// TIA Portal V19 export
DATA_BLOCK "UP_CM03.GP03"   // DB1003
// stored: AutoNumber false, InstanceOfName UP_Spuele.GP0x, InstanceOfType FB
"UP_Spuele.GP0x"
   // VAR RETAIN
   //    In { ExternalAccessible := 'False'; ExternalVisible := 'False'; ExternalWritable := 'False'} : Struct
   //       NotHalt : Bool;
   //       ext_Freigabe : Bool;
   //       TW_senkt : Bool;
   //       Auto : Bool;
   //       Ein : Bool;
   //       FU_betriebsbereit : Bool;
   //       FU_Stoerung : Bool;
   //       Niv_TLS : Bool;
   //       Niv_min : Bool;
   //       Frg_Niv_CM05 : Bool;
   //       SRM_Saugseite_auf : Bool;
   //       SRM_Saugseite_zu : Bool;
   //       SRM_Druckseite_auf : Bool;
   //       SRM_Druckseite_zu : Bool;
   //       GW_p_UP : Bool;
   //       Betriebsart : USInt;
   //       FU_speed : Int;
   //       Druck_Pumpe : Real;
   //    END_STRUCT;
   //    Param { ExternalAccessible := 'False'; ExternalVisible := 'False'; ExternalWritable := 'False'} : Struct
   //       SW_Hand : Int;
   //       SW_Auto_AZ : Int;
   //       SW_Auto_aAZ : Int;
   //       Spülzeit : Time;
   //       DT_Druckaufbau : Time;
   //       DT_Testzeit : Time;
   //       SW_Drucktest : Real;
   //       "Name" : String[12];
   //    END_STRUCT;
   //    Zst { ExternalAccessible := 'False'; ExternalVisible := 'False'; ExternalWritable := 'False'} : Struct
   //       Niveau : USInt;
   //       Status_GP0x : USInt;
   //       Status_DT : USInt;
   //       Restzeit_Spülen : Time;
   //       Restzeit_DT : Time;
   //       TON_Spülventil_auf : Bool;
   //       Spuelen : Bool;
   //       Spuelen_aktiv : Bool;
   //       Drucktest_aktiv : Bool;
   //       Umwaelzen : Bool;
   //       Zeit_laeuft : Bool;
   //       Drucktest_ok : Bool;
   //       Bedienung_erlaubt : Bool;
   //       speed : Int;
   //    END_STRUCT;
   //    Mld { ExternalAccessible := 'False'; ExternalVisible := 'False'; ExternalWritable := 'False'} : Struct
   //       Niv_TLS : Bool;
   //       Niv_Sensorfehler : Bool;
   //       GW_p_UP : Bool;
   //       FU_nicht_bereit : Bool;
   //       FU_Stoerung : Bool;
   //       n_Auto : Bool;
   //       TO_Druckaufbau : Bool;
   //       Drucktest_ok : Bool;
   //       DT_Fehler : Bool;
   //       Pu_Spuelen_Fertig : Bool;
   //    END_STRUCT;
   //    Out { ExternalAccessible := 'False'; ExternalVisible := 'False'; ExternalWritable := 'False'} : Struct
   //       GP0x_Ein : Bool;
   //       Ventil_Saugseite : Bool;
   //       Ventil_Druckseite : Bool;
   //       Spülventil : Bool;
   //       Ventil_CM05 : Bool;
   //       Soll_speed : Int;
   //    END_STRUCT;
   // END_VAR
   // VAR
   //    IEC_Timer { ExternalAccessible := 'False'; ExternalVisible := 'False'; ExternalWritable := 'False'} : Struct
   //       Spülventil_auf { S7_SetPoint := 'True'} : TON_TIME;
   //       Spülen { S7_SetPoint := 'True'} : TP_TIME;
   //       GW_p { S7_SetPoint := 'True'} : TON_TIME;
   //       Drucktest { S7_SetPoint := 'True'} : TP_TIME;
   //       TO_Druckaufbau { S7_SetPoint := 'True'} : TON_TIME;
   //       Ventil_CMO5 { S7_SetPoint := 'True'} : TOF_TIME;
   //    END_STRUCT;
   //    R_TRIG_Hand_EIN { ExternalAccessible := 'False'; ExternalVisible := 'False'; ExternalWritable := 'False'} : R_TRIG;
   // END_VAR
BEGIN
END_DATA_BLOCK
